FUNCTION TryConvert_BOOL_TO_SINT : BOOL
VAR_INPUT
	in : BOOL;
	out : REFERENCE TO SINT;
END_VAR

out := BOOL_TO_SINT(in);
TryConvert_BOOL_TO_SINT := TRUE;

END_FUNCTION

(* stored: Version 1.1.0.1, ProductVersion 3.1.4024.12
   POU TryConvert_BOOL_TO_SINT: Id {bdb07fa9-6bf0-4b02-b1b6-6ba7eaf8c765}, SpecialFunc None *)
